FUNCTION_BLOCK FB_LamparaMemorizada_ST
VAR_INPUT
END_VAR
VAR_OUTPUT
END_VAR
VAR
    Lampara AT %Q*: BOOL;
    PulsadorConexion AT %I*: BOOL;
    PulsadorDesconexion AT %I*: BOOL;
END_VAR

IF PulsadorDesconexion THEN
    Lampara := FALSE
ELSIF PulsadorConexion THEN
    Lampara := TRUE;
END_IF

END_FUNCTION_BLOCK

(* stored: Version 1.1.0.1, ProductVersion 3.1.4024.12
   POU FB_LamparaMemorizada_ST: Id {0354aed3-5461-4991-a04b-d00e3b16aefe}, SpecialFunc None *)
